FUNCTION_BLOCK PUBLIC FB_Machine
VAR_INPUT
	bButton				:	BOOL;
	bInsertCoin			:	BOOL;
	bTakeProduct		:	BOOL;
	bTakeCoin			:	BOOL;
END_VAR
VAR_OUTPUT
	eState 				:	E_States;
	nProducts			:	UINT;
END_VAR
VAR	
	rtrigButton			:	R_TRIG;
	rtrigInsertCoin		:	R_TRIG;
	rtrigTakeProduct	:	R_TRIG;
	rtrigTakeCoin		:	R_TRIG;	
END_VAR

rtrigButton(CLK := bButton);
rtrigInsertCoin(CLK := bInsertCoin);
rtrigTakeProduct(CLK := bTakeProduct);
rtrigTakeCoin(CLK := bTakeCoin);

IF (rtrigButton.Q) THEN
	THIS^.PressButton();
END_IF

IF (rtrigInsertCoin.Q) THEN
	THIS^.InsertCoin();
END_IF

IF (rtrigTakeProduct.Q) THEN
	THIS^.CustomerTakesProduct();
END_IF

IF (rtrigTakeCoin.Q) THEN
	THIS^.CustomerTakesCoin();
END_IF

METHOD INTERNAL CustomerTakesCoin : BOOL
VAR_INPUT
END_VAR
IF (THIS^.eState = E_States.eCoinEjected) THEN
	ADSLOGSTR(ADSLOG_MSGTYPE_HINT, 'Customer has taken the coin.', '');
	eState := E_States.eWaiting;
END_IF
END_METHOD

METHOD INTERNAL CustomerTakesProduct : BOOL
VAR_INPUT
END_VAR
IF (THIS^.eState = E_States.eProductEjected) THEN
	ADSLOGSTR(ADSLOG_MSGTYPE_HINT, 'Customer has taken the product.', '');
	eState := E_States.eWaiting;
END_IF
END_METHOD

METHOD FB_init : BOOL
VAR_INPUT
	bInitRetains : BOOL; // if TRUE, the retain variables are initialized (warm start / cold start)
	bInCopyCode : BOOL;  // if TRUE, the instance afterwards gets moved into the copy code (online change)
	nProducts :	UINT;
END_VAR
THIS^.nProducts := nProducts;
END_METHOD

METHOD INTERNAL InsertCoin : BOOL
VAR_INPUT
END_VAR
IF (THIS^.eState = E_States.eWaiting) THEN
	ADSLOGSTR(ADSLOG_MSGTYPE_HINT, 'Customer has insert a coin.', '');
	THIS^.eState := E_States.eHasCoin;
END_IF
END_METHOD

METHOD INTERNAL PressButton : BOOL
VAR_INPUT
END_VAR
IF (THIS^.eState = E_States.eHasCoin) THEN
	IF (THIS^.nProducts > 0) THEN
		THIS^.nProducts := THIS^.nProducts - 1;
		ADSLOGSTR(ADSLOG_MSGTYPE_HINT, 'Customer has pressed the button. Output product.', '');
		THIS^.eState := E_States.eProductEjected;
	ELSE				
		ADSLOGSTR(ADSLOG_MSGTYPE_HINT, 'Customer has pressed the button. No more products. Return coin.', '');
		THIS^.eState := E_States.eCoinEjected;
	END_IF
END_IF
END_METHOD

END_FUNCTION_BLOCK

(* stored: Version 1.1.0.1, ProductVersion 3.1.4022.12
   POU FB_Machine: Id {c0f33541-2076-46c4-b6c1-6cda993f2079}, SpecialFunc None
   Method CustomerTakesCoin: Id {89905c24-f64a-47f7-9831-f13322442984}
   Method CustomerTakesProduct: Id {864cf179-504e-41f8-bee7-1db8496a9131}
   Method FB_init: Id {206fd956-e051-41c8-9621-20937bbc1327}
   Method InsertCoin: Id {90193e61-c93d-4256-8346-8e010f353619}
   Method PressButton: Id {4dad7645-4644-44fe-b6c3-addd1e666600} *)
